// TwinCAT 3 PLC project Sample04
// ProgramVersion: 3.1.4020.1
// libraries:
//   Tc2_Standard, * (Beckhoff Automation GmbH)
//   Tc2_System, * (Beckhoff Automation GmbH)
//   Tc3_Module, * (Beckhoff Automation GmbH)
// project tree:
//   / PlcTask.TcTTO
//   POUs/ FB_Matrix.TcPOU, MAIN.TcPOU
// real-time tasks:
//   TASK PlcTask: cycle T#10ms, priority 20, ADS port 350

CONFIGURATION Sample04
    RESOURCE PLC ON TwinCAT3
        TASK PlcTask(INTERVAL := T#10ms, PRIORITY := 20);
        PROGRAM MAIN WITH PlcTask : MAIN;
    END_RESOURCE
END_CONFIGURATION

// ---- POUs/MAIN.TcPOU
PROGRAM MAIN
VAR
	fbMatrix			: FB_Matrix;
	arrayA1 			: ARRAY[1..2, 1..2] OF DINT := [1, 2, 3, 4];
	arrayB1 			: ARRAY[1..2, 1..2] OF DINT := [5, 6, 7, 8];
	arrayX1 			: ARRAY[1..2, 1..2] OF DINT;
	
	arrayA2 			: ARRAY[1..3, 1..3] OF DINT := [1, 2, 3, 4, 5, 6, 7, 8, 9];
	arrayB2 			: ARRAY[1..3, 1..3] OF DINT := [5, 6, 7, 8, 10, 11, 12, 13, 14];
	arrayX2 			: ARRAY[1..3, 1..3] OF DINT;				
END_VAR

fbMatrix.Multiplication(arrayA1, arrayB1, arrayX1);

fbMatrix.Multiplication(arrayA2, arrayB2, arrayX2);

END_PROGRAM

// ---- POUs/FB_Matrix.TcPOU
FUNCTION_BLOCK FB_Matrix
VAR_INPUT
END_VAR
VAR_OUTPUT
END_VAR
VAR
END_VAR

METHOD PUBLIC Multiplication : BOOL
VAR_IN_OUT
	arrayA 			: ARRAY[*, *] OF DINT;
	arrayB 			: ARRAY[*, *] OF DINT;
	arrayX 			: ARRAY[*, *] OF DINT;	
END_VAR
VAR
	nIndex1, nIndex2, nIndex3, nIndex4	: DINT;
END_VAR;
FOR nIndex1 := LOWER_BOUND(arrayA, 1) TO UPPER_BOUND(arrayA, 1) DO
	FOR nIndex2 := LOWER_BOUND(arrayB, 2) TO UPPER_BOUND(arrayB, 2) DO
		nIndex4 := 0;
		FOR nIndex3 := LOWER_BOUND(arrayA, 2) TO UPPER_BOUND(arrayA, 2) DO
			nIndex4 := nIndex4 + arrayA[nIndex1, nIndex3] * arrayB[nIndex3, nIndex2];
		END_FOR;
		arrayX[nIndex1, nIndex2] := nIndex4;
	END_FOR;
END_FOR;
END_METHOD

END_FUNCTION_BLOCK
